{attribute 'qualified_only'}
VAR_GLOBAL
	FpistonMainJib : LREAL;
	FpistonBoom : LREAL;
END_VAR

(* stored: Version 1.1.0.1, ProductVersion 3.1.4024.9
   GVL Work: Id {5ed653ee-4ae3-47db-9070-5b8ede254b65} *)
